TYPE "UDT_ZC_RECETA_CIP_DESINF_ENJ"
VERSION : 0.1
   STRUCT
      TiempoEmpujeADestino : Int;   // DESINF ENJ. Tiempo de empuje a destino
      TiempoMaxVaciadoDestino : Int;   // DESINF ENJ. Tiempo Max vaciado destino
      TiempoEmpujeDestinoACIP : Int;   // DESINF ENJ. Tiempoi empuje desde equipo a CIP
      TiempoMaxEnjuague : Int;   // DESINF ENJ. Tiempo Maximo Enjuague
      TiempoEnjuagueConConductividad : Int;   // DESINF ENJ. Tiempo enjuague con conductividad
      ReservaInt_1 : Int;   // DESINF ENJ.
      ReservaInt_2 : Int;   // DESINF ENJ.
      TemperaturaEnjuague : Real;   // DESINF ENJ. Temperatura Enjuague
      TemperaturaHisteresis : Real;   // DESINF ENJ. Temperatura Enjuague Histeresis
      ConductividadDrenaje : Real;   // DESINF ENJ. Conductividad para Drenaje
      ConductividadEnjuagueOk : Real;   // DESINF ENJ. Conductividad para Enjuague OK
      ConductividadDrenajeAguaRecup : Real;   // DESINF ENJ. Conductividad para drenaje/agua recup.
      ProcentajeEnvioDQO : Real;   // DESINF ENJ. Porcentaje de tiempo de envio a DQO
   END_STRUCT;

END_TYPE

